// TIA Portal V20 export
VAR_GLOBAL   // PLC tag table "CentralShifter"
   iCS_SensorHoming_Left AT %I3000.0 : Bool;
   iCS_SensorHoming_Right AT %I3000.2 : Bool;
   CS_R1_Sen_Drv_1 AT %I3100.0 : Bool;
   CS_R1_Sen_Drv_2 AT %I3100.1 : Bool;
   CS_R1_Sen_Drv_3 AT %I3100.2 : Bool;
   CS_R1_Sen_Drv_4 AT %I3100.3 : Bool;
   CS_R1_Sen_Val1_Up AT %I3100.4 : Bool;
   CS_R1_Sen_Val1_Down AT %I3100.5 : Bool;
   CS_R1_Sen_Val2_Up AT %I3100.6 : Bool;
   CS_R1_Sen_Val2_Down AT %I3100.7 : Bool;
   CS_R1_Hyd_Filtr AT %I3101.0 : Bool;
   CS_R1_Hyd_Empty AT %I3101.1 : Bool;
   CS_R1_Safety1_1 AT %I3150.0 : Bool;
   CS_R1_Safety2_1 AT %I3150.1 : Bool;
   CS_R1_Safety3_1 AT %I3150.2 : Bool;
   CS_R1_Safety4_1 AT %I3150.3 : Bool;
   CS_R1_Safety1_2 AT %I3150.4 : Bool;
   CS_R1_Safety2_2 AT %I3150.5 : Bool;
   CS_R1_Safety3_2 AT %I3150.6 : Bool;
   CS_R1_Safety4_2 AT %I3150.7 : Bool;
   CS_R1_Valve_Up AT %Q3100.0 : Bool;
   CS_R1_Valve_Down AT %Q3100.1 : Bool;
   CS_R1_Hydraulic_Unit AT %Q3100.2 : Bool;
   iCS_L_Distance_Value AT %IW3102 : Int;
   CS_R2_Sen_Drv_1 AT %I3200.0 : Bool;
   CS_R2_Sen_Drv_2 AT %I3200.1 : Bool;
   CS_R2_Sen_Drv_3 AT %I3200.2 : Bool;
   CS_R2_Sen_Drv_4 AT %I3200.3 : Bool;
   CS_R2_Sen_Val1_Up AT %I3200.4 : Bool;
   CS_R2_Sen_Val1_Down AT %I3200.5 : Bool;
   CS_R2_Sen_Val2_Up AT %I3200.6 : Bool;
   CS_R2_Sen_Val2_Down AT %I3200.7 : Bool;
   CS_R2_Hyd_Filtr AT %I3201.0 : Bool;
   CS_R2_Hyd_Empty AT %I3201.1 : Bool;
   iCS_R_Distance_Value AT %IW3202 : Int;
   CS_R2_Safety1_1 AT %I3250.0 : Bool;
   CS_R2_Safety2_1 AT %I3250.1 : Bool;
   CS_R2_Safety3_1 AT %I3250.2 : Bool;
   CS_R2_Safety4_1 AT %I3250.3 : Bool;
   CS_R2_Safety1_2 AT %I3250.4 : Bool;
   CS_R2_Safety2_2 AT %I3250.5 : Bool;
   CS_R2_Safety3_2 AT %I3250.6 : Bool;
   CS_R2_Safety4_2 AT %I3250.7 : Bool;
   CS_R2_Valve_Up AT %Q3200.0 : Bool;
   CS_R2_Valve_Down AT %Q3200.1 : Bool;
   CS_R2_Hydraulic_Unit AT %Q3200.2 : Bool;
END_VAR
